RoboDK station: TM12 Workstation.rdk

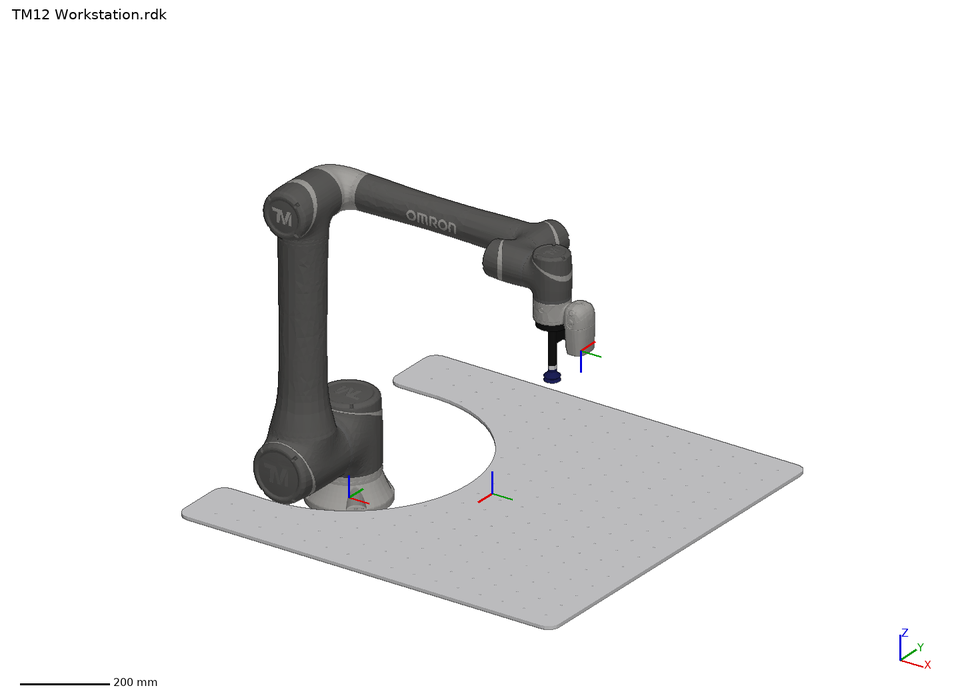
[picture v0: the station drawn from its stored meshes, robots at their saved joint values, targets as dots, program paths as lines]
Station TM12 Station (saved by RoboDK 5.3.5). Poses are relative to the parent item; angles as X-Y-Z fixed-axis rotations.
Station parameters (name, value as stored): IO_1, 1, IO_0, 0
  - frame Omron TM12 Base at (0, 0, -128) mm
    - robot Omron TM12: 6 axes, payload 12 kg, reach 1300 mm, repeatability 0.1 mm, weight 33.3 kg
        modified DH rows (alpha deg, a mm, theta deg, d mm): 0, 0, 0, 165.2; 90, 0, 90, 0; 0, 636.1, 0, 0; 0, 557.9, -90, 156.3; -90, 0, 0, 106; 90, 0, 180, 113.15
        joint limits [-270, -180, -166, -180, -180, -270] to [270, 180, 166, 180, 180, 270]; home [0, 0, 90, -90, 90, 0]; saved at [0, 0, 90, 0, 90, 0]
      - tool TM12 Suction Cup v2, TCP at (0, 0, 146) mm, size 75 x 82.5 x 152 mm, geometry from TM12 Suction Cup v2.step
      - frame Camera Ref at (0, 79, 53) mm
        - camera Camera 1
    - frame Bordet at (392.5, -2.5, 120) mm, rotated rx 0 ry 0 rz -90 deg
      - object Omron TM12 Work Surface v1 at (0, 0, 0) mm, size 1000 x 1025 x 8 mm, geometry from Omron TM12 Work Surface v1.step
